PROGRAM MAIN
VAR
	        PLCVar : ARRAY [0..99] OF INT;
 Index: BYTE;
END_VAR

FOR Index := 0 TO 99 DO
 PLCVar[Index] := 3500 + INDEX;
END_FOR

END_PROGRAM

(* stored: Version 1.1.0.1, ProductVersion 3.1.4024.10
   POU MAIN: Id {a739bf6f-fed5-46b7-bfde-607d16051ca1}, SpecialFunc None *)
